TYPE AxesAzimuthAxisStatuses :
STRUCT
	///Is the axis in a busy state?
	busyStatus: BusyStatus;
	///Is the axis in a healthy state?
	healthStatus: HealthStatus;
	///Is the axis powered on or off?
	poweredStatus: PoweredStatus;
END_STRUCT
END_TYPE

(* stored: Version 1.1.0.1, ProductVersion 3.1.4019.2
   DUT AxesAzimuthAxisStatuses: Id {2f145e82-c1fc-4911-a277-d465341e463d} *)
